Fanuc KAREL source: ko00044.KL

-- PROVISIONAL review KL for V770-1; original PC SHA256 5f18ea7c4d2e55651e5d3f080668c318c84aa9ee18d1e23cd2981b382742a3f0
-- Incomplete behavior may be omitted. Consult companion uncertainty JSON. Do not deploy.
PROGRAM KO00044
%NOLOCKGROUP
BEGIN
  -- UNRESOLVED_PC offsets 5-12; opcodes 9D,23
  -- UNRESOLVED_PC offsets 17-69; opcodes 27,27,49,7E,AD,27,49,7E,AD,22,31,7E,4A
  -- UNRESOLVED_PC offsets 74-78; opcodes 7F
END KO00044
